// TIA Portal V17 export
// export: Created 2022-07-20T06:59:44.0018143Z, ExportSetting WithDefaults, DisplayName Totally Integrated Automation Portal, DisplayVersion V17, DisplayName TIA Portal Openness, DisplayVersion V17, DisplayName TIA Portal Version Control Interface, DisplayVersion V17, DisplayName SINAMICS Startdrive Advanced, DisplayVersion V17, DisplayName SINAMICS Startdrive G130, G150, S120, S150, SINAMICS MV, S210, DisplayVersion V17, DisplayName SINAMICS Startdrive G110M, G120, G120C, G120D, G120P, G115D, DisplayVersion V17, DisplayName STEP 7 Professional, DisplayVersion V17, DisplayName STEP 7 Safety, DisplayVersion V17, DisplayName WinCC Advanced, DisplayVersion V17
FUNCTION "FC10070_ScalingAirExtraction" : Void   // FC10070, LAD
TITLE = FC10070_ScalingAirExtraction
{ S7_Optimized_Access := 'TRUE' }
AUTHOR : Jonathan
FAMILY : 1007x_DRYER_UV
VERSION : 1.1
// Release note : 
// 1.0 - Version alphahet, only analog output
// 1.1 - Iris improvment : add percentage value to be reeuse for PWM control
// stored: AutoNumber false, IsIECCheckEnabled false, SetENOAutomatically false, UDAEnableTagReadback false
   VAR_INPUT
      SetPoint : Real;
      X_UVPower_Min : Real;   // 0-100%
      X_UVPower_Max : Real;   // 0-100%
      Y_AirPower_Min : Real;   // 0-100%
      Y_AirPower_Max : Real;   // 0-100%
      PWM_Minimum : Real;   // Frequence
      PWM_Maximum : Real;   // Frequence
   END_VAR
   VAR_OUTPUT
      AnalogValue : Int;
      PwmFrequenceValue : Real;
   END_VAR
   VAR_TEMP
      SetPointNorm : Real;
      Y_AirPower_Min_Analog : Real;   // Y_AirPower_Min/(27648/100)
      Y_AirPower_Max_Analog : Real;   // Y_AirPower_Max/(27648/100)
      Y_AirPower_Min_PWM : Real;   // Y_AirPower_Min/(PWM_Max-PWM_Min) + PWM_Min
      Y_AirPower_Max_PWM : Real;   // Y_AirPower_Max/(PWM_Max-PWM_Min) + PWM_Min
      Percentage_to_Pwm : Real;   // 1% = x Hz
   END_VAR
BEGIN

REGION Network 1: Normalize the set point
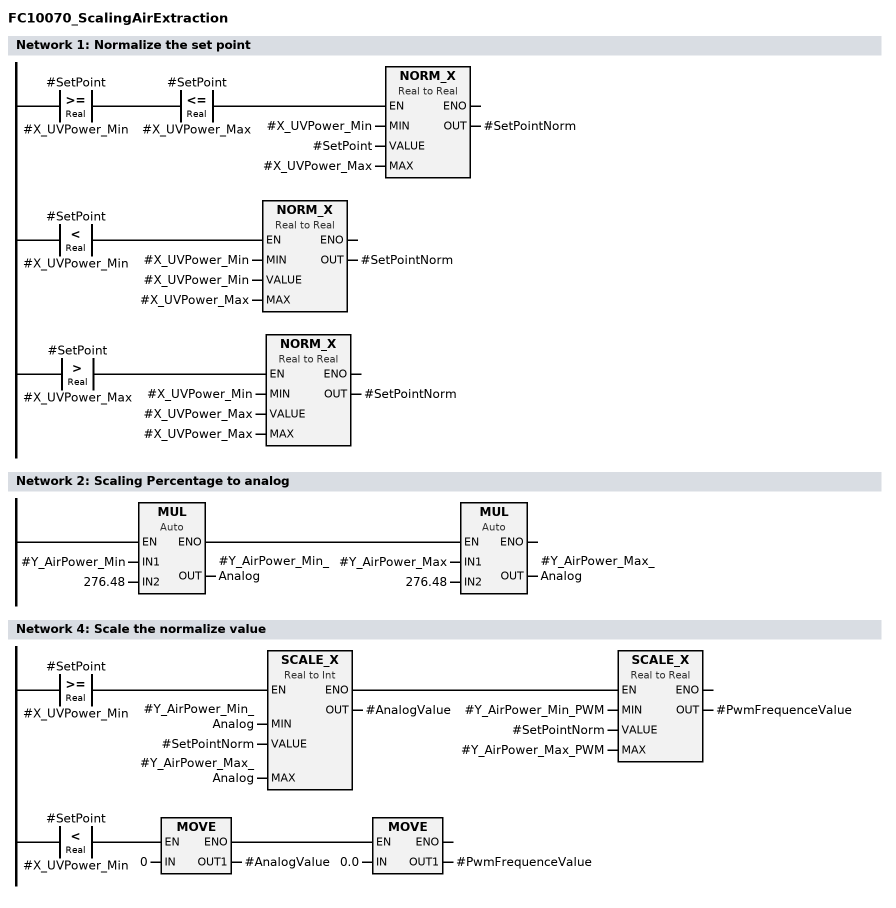
   RUNG wire#powerrail
      { S7_Templates := "SrcType := Real" } GE_Contact(in1 := #SetPoint, in2 := #X_UVPower_Min)
      { S7_Templates := "SrcType := Real" } LE_Contact(in1 := #SetPoint, in2 := #X_UVPower_Max)
      { S7_Templates := "[SrcType := Real, DestType := Real]" } Normalize(min := #X_UVPower_Min, value := #SetPoint, max := #X_UVPower_Max, out => #SetPointNorm)
   END_RUNG
   RUNG wire#powerrail
      { S7_Templates := "SrcType := Real" } LT_Contact(in1 := #SetPoint, in2 := #X_UVPower_Min)
      { S7_Templates := "[SrcType := Real, DestType := Real]" } Normalize(min := #X_UVPower_Min, value := #X_UVPower_Min, max := #X_UVPower_Max, out => #SetPointNorm)
   END_RUNG
   RUNG wire#powerrail
      { S7_Templates := "SrcType := Real" } GT_Contact(in1 := #SetPoint, in2 := #X_UVPower_Max)
      { S7_Templates := "[SrcType := Real, DestType := Real]" } Normalize(min := #X_UVPower_Min, value := #X_UVPower_Max, max := #X_UVPower_Max, out => #SetPointNorm)
   END_RUNG
   // the same network as SCL:
   IF (#SetPoint >= #X_UVPower_Min) AND (#SetPoint <= #X_UVPower_Max) THEN
       #SetPointNorm := NORM_X(MIN := #X_UVPower_Min, VALUE := #SetPoint, MAX := #X_UVPower_Max);
   END_IF;
   IF #SetPoint < #X_UVPower_Min THEN
       #SetPointNorm := NORM_X(MIN := #X_UVPower_Min, VALUE := #X_UVPower_Min, MAX := #X_UVPower_Max);
   END_IF;
   IF #SetPoint > #X_UVPower_Max THEN
       #SetPointNorm := NORM_X(MIN := #X_UVPower_Min, VALUE := #X_UVPower_Max, MAX := #X_UVPower_Max);
   END_IF;
END_REGION

REGION Network 2: Scaling Percentage to analog
   RUNG wire#powerrail
      { S7_GenerateENO := "TRUE" } Mul(in1 := #Y_AirPower_Min, in2 := 276.48, out => #Y_AirPower_Min_Analog)
      { S7_GenerateENO := "TRUE" } Mul(in1 := #Y_AirPower_Max, in2 := 276.48, out => #Y_AirPower_Max_Analog)
   END_RUNG
   // the same network as SCL:
   // ENO of a box is taken as its EN; it also drops when the box reports an error
   #Y_AirPower_Min_Analog := #Y_AirPower_Min * 276.48;
   #Y_AirPower_Max_Analog := #Y_AirPower_Max * 276.48;
END_REGION

REGION Network 3 (SCL): Y_AirPower_Min/(PWM_Max-PWM_Min) + PWM_Min
   #Percentage_to_Pwm := (#PWM_Maximum - #PWM_Minimum) / 100.0;

   IF #Percentage_to_Pwm > 1 THEN
       #Y_AirPower_Min_PWM := (#Y_AirPower_Min * #Percentage_to_Pwm) + #PWM_Minimum;
       #Y_AirPower_Max_PWM := (#Y_AirPower_Max * #Percentage_to_Pwm) + #PWM_Minimum;
   END_IF;
END_REGION

REGION Network 4: Scale the normalize value
   RUNG wire#powerrail
      { S7_Templates := "SrcType := Real" } GE_Contact(in1 := #SetPoint, in2 := #X_UVPower_Min)
      { S7_Templates := "[SrcType := Real, DestType := Int]" } Scale(min := #Y_AirPower_Min_Analog, value := #SetPointNorm, max := #Y_AirPower_Max_Analog, out => #AnalogValue)
      { S7_Templates := "[SrcType := Real, DestType := Real]"; S7_GenerateENO := "TRUE" } Scale(min := #Y_AirPower_Min_PWM, value := #SetPointNorm, max := #Y_AirPower_Max_PWM, out => #PwmFrequenceValue)
   END_RUNG
   RUNG wire#powerrail
      { S7_Templates := "SrcType := Real" } LT_Contact(in1 := #SetPoint, in2 := #X_UVPower_Min)
      { S7_GenerateENO := "TRUE" } Move(in := 0, out1 => #AnalogValue)
      { S7_GenerateENO := "TRUE" } Move(in := 0.0, out1 => #PwmFrequenceValue)
   END_RUNG
   // the same network as SCL:
   // ENO of a box is taken as its EN; it also drops when the box reports an error
   IF #SetPoint >= #X_UVPower_Min THEN
       #AnalogValue := SCALE_X(MIN := #Y_AirPower_Min_Analog, VALUE := #SetPointNorm, MAX := #Y_AirPower_Max_Analog);
       #PwmFrequenceValue := SCALE_X(MIN := #Y_AirPower_Min_PWM, VALUE := #SetPointNorm, MAX := #Y_AirPower_Max_PWM);
   END_IF;
   IF #SetPoint < #X_UVPower_Min THEN
       #AnalogValue := 0;
       #PwmFrequenceValue := 0.0;
   END_IF;
END_REGION
END_FUNCTION
